{attribute 'qualified_only'}
VAR_GLOBAL
	fbBasetest					: FB_Base;
	
	fbPB1_Wyk1_K1				: FB_Component;
	fbPB1_Wyk1_K2				: FB_Component;
	fbPB1_Wyk1					: FB_ControlElement (fbPB1_Wyk1_K1, fbPB1_Wyk1_K2);
	
	fbPB1_Wyk2_K1				: FB_Component;
	fbPB1_Wyk2_K2				: FB_Component;
	fbPB1_Wyk2					: FB_ControlElement_1 (fbPB1_Wyk2_K1, fbPB1_Wyk2_K2);

	fbPB1_ZL1_Wyk1_K1			: FB_Component;
	fbPB1_ZL1_Wyk1_K2			: FB_Component;
	fbPB1_ZL1_Wyk1				: FB_ControlElement (fbPB1_ZL1_Wyk1_K1, fbPB1_ZL1_Wyk1_K2);
	fbPB1_ZL1_Wyk2_K1			: FB_Component;
	fbPB1_ZL1_Wyk2_K2			: FB_Component;
	fbPB1_ZL1_Wyk2				: FB_ControlElement (fbPB1_ZL1_Wyk2_K1, fbPB1_ZL1_Wyk2_K2);
	fbPB1_ZL1_K1				: FB_Component;
	fbPB1_ZL1_K2				: FB_Component;
	fbPB1_ZL1					: FB_GroupElement (fbPB1_ZL1_Wyk1, fbPB1_ZL1_Wyk2, fbPB1_ZL1_K1, fbPB1_ZL1_K2);
	
	fbPB1_K1					: FB_Component;
	fbPB1_K2					: FB_Component;
	fbPB1_K3					: FB_Component;
	
	fbPB1						: FB_TopElement (fbPB1_Wyk1, fbPB1_Wyk2, fbPB1_ZL1, fbPB1_K1, fbPB1_K2, fbPB1_K3);
	
END_VAR

(* stored: Version 1.1.0.1, ProductVersion 3.1.4024.15
   GVL GVL_Variable: Id {56e59208-4bbf-49fc-a1d8-9f400ac97c02} *)
